(* IEC 61131-3 sources: repolevel_ST_code_completion/output/0127完整版本_带planner/repoeval_PID_controller/readful_result_no_provide, 4 files *)

(* ---- HeatExchanger.st ---- *)
VAR
	now: TIME;
	lastTime: TIME;
	lastPV: REAL := 140;
	A: REAL;
	B: REAL;
	delta_t: REAL;
	SampleTimeSec: REAL;
	DeadTimeIndex: INT;
	DelayQueue: ARRAY[0..99] OF REAL; // Circular buffer for delay
	QueueHead: INT := 0;
	QueueTail: INT := 0;
	QueueSize: INT := 100;
	QueueCount: INT := 0;
	DelayedCO: REAL := 0.0;
END_VAR

now := TIME();
IF ((now - lastTime) > Sample_time) THEN
delta_t := TIME_TO_REAL(Sample_time) / 1000.0; // Convert milliseconds to seconds
  SampleTimeSec := delta_t;

	IF Dead_t <= SampleTimeSec THEN
		DelayedCO := CO; // Skip delay if Dead_t is less than or equal to Sample_time
	ELSE
		DeadTimeIndex := REAL_TO_INT(Dead_t / SampleTimeSec);

		// Store CO in delay queue
		DelayQueue[QueueHead] := CO;
		QueueHead := (QueueHead + 1) MOD QueueSize;
		IF QueueCount < QueueSize THEN
			QueueCount := QueueCount + 1;
		ELSE
			QueueTail := (QueueTail + 1) MOD QueueSize;
		END_IF;

		// Retrieve delayed CO from queue
		IF QueueCount > DeadTimeIndex THEN
			DelayedCO := DelayQueue[(QueueTail + DeadTimeIndex) MOD QueueSize];
		ELSE
			DelayedCO := 0.0; // Default value if delay queue is not yet filled
		END_IF;
	END_IF;

	A := EXP(-delta_t / Tp);
	B := 1 - A;

	PV := A * lastPV + B * Kp * DelayedCO + C;
	lastPV := PV;
	lastTime := now;
END_IF;
END_FUNCTION_BLOCK

(* ---- HeatExchanger2.st ---- *)
VAR
	now: TIME;
	lastTime: TIME := T#0s;
	delta_t: REAL;
	heat_flow: REAL;
	lastTemp: REAL;
	temp_diff: REAL;
	temp_change_rate: REAL;
	temp_change: REAL;
END_VAR

VAR CONSTANT
	millis: REAL := 1000;
END_VAR

now := TIME();
IF ((now - lastTime) > Sample_time) THEN
	// Step 1: Calculate temperature difference
	temp_diff := Temp_Out - Temp_In;

	// Step 2: Calculate heat transfer rate
	heat_flow := Heat_In - (U * temp_diff);

	// Step 3: Calculate temperature change rate
delta_t := TIME_TO_REAL(Sample_time) / millis;
	temp_change_rate := heat_flow / TC;

	// Step 4: Calculate temperature change for the current sampling period
	temp_change := temp_change_rate * delta_t;

	// Step 5: Update room temperature
	Temp := Temp_In + temp_change;

	// Update lastTime and lastTemp
	lastTime := now;
	lastTemp := Temp;
END_IF;
END_FUNCTION_BLOCK

(* ---- PID_controller.st ---- *)
VAR
    e: REAL; // Error
    deltaPV: REAL; // Change in process variable
    SampleTimeSec: REAL; // Sample time in seconds
    CO_temp: REAL; // Temporary control output
END_VAR

// Convert SampleTime from TIME to seconds
SampleTimeSec := TIME_TO_REAL(SampleTime) / millis;

// Step 1: Calculate error
e := SP - PV;

// Step 2: Calculate proportional term
CO_P := Kc * e;

// Step 3: Update and limit integral term
CO_I := CO_I + (Kc * e * (SampleTimeSec / Ti));
IF CO_I > UpperLimit THEN
    CO_I := UpperLimit;
ELSIF CO_I < LowerLimit THEN
    CO_I := LowerLimit;
END_IF

// Step 4: Calculate derivative term
deltaPV := 0; // As 'lastTime' is not defined, no valid derivative can be computed
CO_D := 0;    // Set derivative term to 0

// Step 5: Calculate total control output and limit it
CO_temp := CO_P + CO_I + CO_D;
IF CO_temp > UpperLimit THEN
    CO := UpperLimit;
ELSIF CO_temp < LowerLimit THEN
    CO := LowerLimit;
ELSE
    CO := CO_temp;
END_IF

// Step 6: Save current PV for next cycle
// Removed assignment to undefined variable 'lastTime'
END_FUNCTION_BLOCK

(* ---- Tank.st ---- *)
VAR
  now: TIME;
  lastTime: TIME := T#0ms;
  timeDelta: REAL;
  volumeIn: REAL;
  volumeOut: REAL;
END_VAR
// Step 1: Calculate time delta in seconds
now := TIME();
timeDelta := TIME_TO_REAL(now - lastTime) / 1000.0;

// Step 2: Calculate volume change due to input flow
volumeIn := timeDelta * Process_In;

// Step 3: Calculate volume change due to output flow
volumeOut := timeDelta * Process_Out;

// Step 4: Update tank level
Level := Level + volumeIn - volumeOut;

// Step 5: Constrain tank level within limits
IF Level < Lower_limit THEN
  Level := Lower_limit;
ELSIF Level > Upper_limit THEN
  Level := Upper_limit;
END_IF;

// Update lastTime for the next cycle
lastTime := now;
